{attribute addProperty BoxType "EL4112--0000"}
{attribute addProperty Id "ChannelAT %Q*ARRAY[0..1] OF Channel_969D8B6C3240WcStateAT %I*WcState_64F6A8C6810InfoDataAT %I*InfoData_BC63D37F80100"}
{attribute addProperty CRC "4266795651"}
{attribute addProperty SizeInBites "120"}
{attribute addProperty SizeInBytes "15"}
TYPE EL4112_4AB99AE0 :
STRUCT
	{attribute addProperty Name "Channel"}
	Channel : ARRAY[0..1] OF Channel_969D8B6C;
	{attribute addProperty Name "WcState"}
	WcState : WcState_64F6A8C6;
	{attribute addProperty Name "InfoData"}
	InfoData : InfoData_BC63D37F;
END_STRUCT
END_TYPE

(* stored: Version 1.2.0.0, ProductVersion 3.1.4024.9
   DUT EL4112_4AB99AE0: Id {69e4ea92-cd92-482b-9e90-169cacbd96f9} *)
